FUNCTION_BLOCK FB_L7NHA EXTENDS ZigaLibs_Core.FB_HasInstanceNameAndPath

VAR_INPUT
	bEnable					: BOOL;	// Enable axis
	bReset					: BOOL;	// Reset if an eror is present
	bHalt					: BOOL; // Halts current operation - after setting this to FALSE previous operation is continuoued
	bQuickStop				: BOOL;	// Drive will execute a quick stop
	
	nAcceleration			: UDINT;	// Axis acceleration in UU/s^2
	nDeceleration			: UDINT;	// Axis deceleration in UU/s^
	
	eModeOfOperation		: E_L7NHA_ModeOfOperation;	// Mode of operation
	
	stVelocityCommands		: ST_L7NHA_VelocityCommands;		// Velocity commands when in profile velocity mode
	stPositioningCommands	: ST_L7NHA_PositioningCommands;		// Positioning commands when in profile position mode
	stHomingCommands		: ST_L7NHA_HomingCommands;			// Homing commands when in homing sequence
	stProfileTorqueCommands	: ST_L7NHA_ProfileTorqueCommands;	// Profile torque commands when using Profile Torque mode
	
	fRatedTorque			: REAL; // Rated torque in mNm - required for torque calculation

	stUserUnitParameters	: ST_L7NHA_UserUnitParams;
END_VAR

VAR_OUTPUT
	eAxisState			: E_L7NHA_DriveState;	// Axis state, actual state reported back from drive
	
	eErrorCode			: E_L7NHA_ErrorId;	// Error code, if drive is in fault state
	
	bHomingRequired		: BOOL;	// If homing is required, this flag will be set to true (usually after a power reset)
	
	bMovingPositive		: BOOL;	// Indicating axis is rotating in positive direction
	bMovingNegative		: BOOL;	// Indicating axis is rotating in negative direction
	
	stPositioningStatus	: ST_L7NHA_PositioningStatus;	// Status of the positioning procedure - only valid when in positioning mode
	stHomingStatus		: ST_L7NHA_HomingStatus;		// Status of the homing procedure - only valid when in homing mode
	
	fCalculatedActualTorque	: REAL;
	fCalculatedTargetTorque	: REAL;
	
	eActualModeOfOperation	: E_L7NHA_ModeOfOperation;
	stMotionFeedback		: ST_L7NHA_MotionFeedback;	// Motion feedback from the drive

	stDigitalInputs	:		 ST_L7NHA_DigitalInputs;
	
	bModeOfOperationNotImplemented	: BOOL;	// Will be TRUE if the selected mode of operation is not implemented (axis has to be in enabled state for this flag to be valid!)
END_VAR

// Local variables
VAR
	eAxisStateInternal		: E_L7NHA_DriveState;
	stDataToDriveInternal	: ST_L7NHA_DataToDrive;
	TonCommandTimeout		: Tc2_Standard.TON := (PT := T#1S);
	RtrigMoveToPosition		: Tc2_Standard.R_TRIG;
	RtrigStartHoming		: Tc2_Standard.R_TRIG;
	nPreviousPosition		: DINT;
	RtrigResetTrigger		: Tc2_Standard.R_TRIG;
	RtrigHomingFinished		: Tc2_Standard.R_TRIG;
	TonMotorMovingStatusValid	: Tc2_Standard.TON;
	RtrigModeOfOperationNotImplemented	: Tc2_Standard.R_TRIG;
	eModeOfOpereationOld		: E_L7NHA_ModeOfOperation;
	_logger					: REFERENCE TO ZigaLibs_Logging.I_Logger;
	_sb						: ZigaLibs_Core.FB_StringBuilder;
END_VAR

// IO
VAR
	stDataFromDrive	AT %I* : ST_L7NHA_DataFromDrive;
	stDataToDrive	AT %Q* : ST_L7NHA_DataToDrive;
	stEthercatInfo	AT %I* : ST_L7NHA_EthercatData;
END_VAR

// Sometimes axis wont go to enabled - in that case a timeout should be triggered
TonCommandTimeout(in := eAxisStateInternal = E_L7NHA_DriveState.OPERATION_ENABLED);
// Reset triggering
RtrigResetTrigger(CLK := bReset);


// Abs encoder value is not valid if bit 14 is FALSE (homing has not been completed yet after a power reset/encoder error)
bHomingRequired := stDataFromDrive.StatusWord.14 = FALSE;

// Calling halt will overwrite this - to enable automatic clearing, setting it to false by default
stDataToDriveInternal.ControlWord.8 := FALSE;

// State machine based on the drive's feedback
eAxisStateInternal := THIS^.GetDriveState();

bModeOfOperationNotImplemented := FALSE;
		
// State machine based on actual state reported back from the drive
CASE eAxisStateInternal OF
	E_L7NHA_DriveState.SWITCH_ON_DISABLED:	
		IF bEnable THEN
			Shutdown();
		ELSE
			DisableVoltage();
		END_IF
	
	E_L7NHA_DriveState.READY_TO_SWITCH_ON:
		IF NOT TonCommandTimeout.Q THEN
			SwitchOnEnableOperation();
		END_IF
		
	E_L7NHA_DriveState.OPERATION_ENABLED:
		TonCommandTimeout.IN := FALSE;
		SwitchOnEnableOperation();

		// Execute different mode based on mode of operation setting
		CASE eModeOfOperation OF
			E_L7NHA_ModeOfOperation.PROFILE_POSITION:
				ProfilePosition();
				
			E_L7NHA_ModeOfOperation.PROFILE_VELOCITY:
				ProfileVelocity();
				
			E_L7NHA_ModeOfOperation.HOMING:
				Homing();
				
			E_L7NHA_ModeOfOperation.PROFILE_TORQUE:
				ProfileTorque();
				
			ELSE
				bModeOfOperationNotImplemented := TRUE;
				IF eModeOfOperation <> eModeOfOpereationOld THEN
					IF __ISVALIDREF(_logger) THEN
						_logger.LogError(_sb.Reset()
							.AddString('L7NHA axis ')
							.AddWithDblQuotationMarks(THIS^.InstanceName)
							.AddString(': Mode of operation is not supported! Selected mode is ')
							.AddWithDblQuotationMarks(TO_STRING(eModeOfOperation)));
					END_IF
				END_IF
		END_CASE
		
	E_L7NHA_DriveState.FAULT:
		IF RtrigResetTrigger.Q THEN
			FaultReset();
		ELSE
			stDataToDriveInternal.ControlWord.7 := FALSE;
		END_IF
	
END_CASE

// Override any command if enable is false (transitioning states) - exception is fault, where reset needs to be sent
IF NOT bEnable AND eAxisStateInternal <> E_L7NHA_DriveState.FAULT THEN
	DisableVoltage();
END_IF

// Halt - has a different meaning in PP,PV or homing 
// Usally it "pauses" the current procedure and after halt is set to FALSE drive will proceed where it left off
IF bHalt THEN
	Halt();
END_IF

// Quick stop
IF bQuickStop THEN
	stDataToDriveInternal.ControlWord.1 := bQuickStop;
	stDataToDriveInternal.ControlWord.2 := NOT bQuickStop;
END_IF

// Setting acceleration/deceleration always
stDataToDriveInternal.ProfileAcceleration := nAcceleration;
stDataToDriveInternal.ProfileDeceleration := nDeceleration;

// Mode of operation
stDataToDriveInternal.ModeOfOperation := eModeOfOperation;


// =======================================================================
// ==================== SETTING FB OUTPUTS ===============================
// =======================================================================

// Axis state
eAxisState := eAxisStateInternal;

// Overwriting status for positioning/homing if not in that mode
// Clear homing status if not in that mode
IF eModeOfOperation <> E_L7NHA_ModeOfOperation.HOMING THEN
	MEMSET(
		destAddr := ADR(stHomingStatus),
		n := SIZEOF(stHomingStatus),
		fillByte := 0);
END_IF
 
// Clear positioning status if not in that mode
IF eModeOfOperation <> E_L7NHA_ModeOfOperation.PROFILE_POSITION THEN
	MEMSET(
		destAddr := ADR(stPositioningStatus),
		n := SIZEOF(stPositioningStatus),
		fillByte := 0);
END_IF

// Motion status
TonMotorMovingStatusValid(
	IN := nPreviousPosition <> stDataFromDrive.MotionFeedback.ActualPosition,
	PT := T#30MS);

bMovingPositive := (nPreviousPosition < stDataFromDrive.MotionFeedback.ActualPosition) AND TonMotorMovingStatusValid.Q;
bMovingNegative := (nPreviousPosition > stDataFromDrive.MotionFeedback.ActualPosition) AND TonMotorMovingStatusValid.Q;
nPreviousPosition := stDataFromDrive.MotionFeedback.ActualPosition;

// Digital inputs mapping
stDigitalInputs.NOT_SW := stDataFromDrive.DigitalInputs.0;
stDigitalInputs.POT_SW := stDataFromDrive.DigitalInputs.1;
stDigitalInputs.DI1_OPEN := stDataFromDrive.DigitalInputs.16;
stDigitalInputs.DI2_OPEN := stDataFromDrive.DigitalInputs.17;
stDigitalInputs.DI3_OPEN := stDataFromDrive.DigitalInputs.18;
stDigitalInputs.DI4_OPEN := stDataFromDrive.DigitalInputs.19;
stDigitalInputs.DI5_OPEN := stDataFromDrive.DigitalInputs.20;
stDigitalInputs.DI6_OPEN := stDataFromDrive.DigitalInputs.21;
stDigitalInputs.DI7_OPEN := stDataFromDrive.DigitalInputs.22;
stDigitalInputs.DI8_OPEN := stDataFromDrive.DigitalInputs.23;
stDigitalInputs.STO_OPEN := stDataFromDrive.DigitalInputs.31;

// Error code
IF eErrorCode <> stDataFromDrive.ErrorCode THEN
	IF __ISVALIDREF(_logger) THEN
		IF stDataFromDrive.ErrorCode = E_L7NHA_ErrorId.NO_ERROR THEN
			_logger.LogInfo(_sb.Reset()
				.AddString('L7NHA axis ')
				.AddWithDblQuotationMarks(THIS^.InstanceName)
				.AddString(' error no longer active.')
				.Create());
		ELSE
			_logger.LogError(_sb.Reset()
				.AddString('L7NHA axis ')
				.AddWithDblQuotationMarks(THIS^.InstanceName)
				.AddString(' error active! Error code: ')
				.AddString(TO_STRING(stDataFromDrive.ErrorCode))
				.AddString(' !')
				.Create());
		END_IF
	END_IF
END_IF

eErrorCode := stDataFromDrive.ErrorCode;

// Motion feedback from drive
stMotionFeedback := stDataFromDrive.MotionFeedback;
// Convert position/velocity to custom units

stMotionFeedback := stDataFromDrive.MotionFeedback;

fCalculatedActualTorque := CalculateTorque(fRatedTorque := fRatedTorque, nDriveTorqueFeedback := stDataFromDrive.MotionFeedback.ActualTorque);
fCalculatedTargetTorque := CalculateTorque(fRatedTorque := fRatedTorque, nDriveTorqueFeedback := stDataFromDrive.MotionFeedback.TargetTorque);

// Actual mode of operation, read from the drive
eActualModeOfOperation := stDataFromDrive.ModeOfOperation;

eModeOfOpereationOld := eModeOfOperation;

// =======================================================================
// ==================== SETTING OUTPUT STRUCTURE TO DRIVE ================
// =======================================================================
stDataToDrive := stDataToDriveInternal;

METHOD PRIVATE CalculateTorque : REAL
VAR_INPUT
	fRatedTorque 			: REAL; // Rated torque in mNm
	nDriveTorqueFeedback 	: INT;	// Drives feedback (0.1% increments, -100%...+100%)
END_VAR
CalculateTorque := fRatedTorque * TO_REAL(nDriveTorqueFeedback);
END_METHOD

METHOD PRIVATE DisableVoltage
stDataToDriveInternal.controlWord := 0;
END_METHOD

METHOD PRIVATE EnableOperation
stDataToDriveInternal.controlWord.0 := 0;
stDataToDriveInternal.controlWord.1 := 1;
stDataToDriveInternal.controlWord.2 := 1;
stDataToDriveInternal.controlWord.3 := 0;
stDataToDriveInternal.controlWord.4 := 0;
stDataToDriveInternal.controlWord.5 := 0;
stDataToDriveInternal.controlWord.6 := 0;
stDataToDriveInternal.controlWord.7 := 0;
END_METHOD

METHOD PRIVATE FaultReset
IF stDataToDriveInternal.controlWord.7 = 0 THEN
	stDataToDriveInternal.controlWord.7 := 1;
	stDataToDriveInternal.controlWord.0 := 0;
	stDataToDriveInternal.controlWord.1 := 0;
	stDataToDriveInternal.controlWord.2 := 0;
	stDataToDriveInternal.controlWord.3 := 0;
END_IF
END_METHOD

METHOD FB_init : BOOL
VAR_INPUT
	bInitRetains : BOOL; // if TRUE, the retain variables are initialized (warm start / cold start)
	bInCopyCode : BOOL;  // if TRUE, the instance afterwards gets moved into the copy code (online change)
	logger		: REFERENCE TO ZigaLibs_Logging.I_Logger; // If you do not want logging, simply set this variable to 0, internal checks will ommit any logging.		
END_VAR
_logger REF= logger;
END_METHOD

// Converts status word to a readable drive state enum
METHOD PRIVATE GetDriveState : E_L7NHA_DriveState
//================ SWITCH_ON_DISABLED =====================
IF stDataFromDrive.StatusWord.0 = FALSE AND
    stDataFromDrive.StatusWord.1 = FALSE AND
    stDataFromDrive.StatusWord.2 = FALSE AND
    stDataFromDrive.StatusWord.3 = FALSE AND
    stDataFromDrive.StatusWord.5 = TRUE AND 
    stDataFromDrive.StatusWord.6 = TRUE
THEN
	GetDriveState := E_L7NHA_DriveState.SWITCH_ON_DISABLED;

//================ READY_TO_SWITCH_ON =====================	
ELSIF stDataFromDrive.StatusWord.0 = TRUE AND
   	   stDataFromDrive.StatusWord.1 = FALSE AND
       stDataFromDrive.StatusWord.2 = FALSE AND
       stDataFromDrive.StatusWord.3 = FALSE AND
       stDataFromDrive.StatusWord.5 = TRUE AND 
       stDataFromDrive.StatusWord.6 = FALSE
THEN
	GetDriveState := E_L7NHA_DriveState.READY_TO_SWITCH_ON;	

//================ SWITCHED_ON ==========================	
ELSIF stDataFromDrive.StatusWord.0 = TRUE AND
   	   stDataFromDrive.StatusWord.1 = TRUE AND
       stDataFromDrive.StatusWord.2 = FALSE AND
       stDataFromDrive.StatusWord.3 = FALSE AND
       stDataFromDrive.StatusWord.5 = TRUE AND 
       stDataFromDrive.StatusWord.6 = FALSE
THEN
	GetDriveState := E_L7NHA_DriveState.SWITCHED_ON;

//================ OPERATION_ENABLED =====================	
ELSIF stDataFromDrive.StatusWord.0 = TRUE AND
   	   stDataFromDrive.StatusWord.1 = TRUE AND
       stDataFromDrive.StatusWord.2 = TRUE AND
       stDataFromDrive.StatusWord.3 = FALSE AND
       stDataFromDrive.StatusWord.5 = TRUE AND 
       stDataFromDrive.StatusWord.6 = FALSE
THEN
	GetDriveState := E_L7NHA_DriveState.OPERATION_ENABLED;

//================ FAULT_REACTION_ACTIVE =====================		
ELSIF stDataFromDrive.StatusWord.0 = TRUE AND
   	   stDataFromDrive.StatusWord.1 = TRUE AND
       stDataFromDrive.StatusWord.2 = TRUE AND
       stDataFromDrive.StatusWord.3 = TRUE AND
       stDataFromDrive.StatusWord.5 = TRUE AND 
       stDataFromDrive.StatusWord.6 = FALSE
THEN
	GetDriveState := E_L7NHA_DriveState.FAULT_REACTION_ACTIVE;

//================ FAULT =====================	
ELSIF  stDataFromDrive.StatusWord.0 = FALSE AND
   	   stDataFromDrive.StatusWord.1 = FALSE AND
       stDataFromDrive.StatusWord.2 = FALSE AND
       stDataFromDrive.StatusWord.3 = TRUE AND 
       stDataFromDrive.StatusWord.6 = FALSE
THEN
	GetDriveState := E_L7NHA_DriveState.FAULT;				
END_IF
END_METHOD

// Halts the axis for as long as called
METHOD PRIVATE Halt : BOOL
VAR_INPUT
END_VAR
stDataToDriveInternal.ControlWord.8 := TRUE;
END_METHOD

ACTION Homing:
// Set the status of homing

// Hooming is in progress
stHomingStatus.InProgress := 
stDataFromDrive.StatusWord.10 = FALSE AND
stDataFromDrive.StatusWord.12 = FALSE AND
stDataFromDrive.StatusWord.13 = FALSE;

// Homing is not started
stHomingStatus.NotStarted := 
stDataFromDrive.StatusWord.10 = TRUE AND
stDataFromDrive.StatusWord.12 = FALSE AND
stDataFromDrive.StatusWord.13 = FALSE;	

// Target not reached	
stHomingStatus.TargetNotReached := 
stDataFromDrive.StatusWord.10 = FALSE AND
stDataFromDrive.StatusWord.12 = TRUE AND
stDataFromDrive.StatusWord.13 = FALSE;

// Homing completed
stHomingStatus.Completed := 
stDataFromDrive.StatusWord.10 = TRUE AND
stDataFromDrive.StatusWord.12 = TRUE AND
stDataFromDrive.StatusWord.13 = FALSE;

// Error - speed is not zero ????
stHomingStatus.ErrorSpeedNotZero := 
stDataFromDrive.StatusWord.10 = FALSE AND
stDataFromDrive.StatusWord.12 = FALSE AND
stDataFromDrive.StatusWord.13 = TRUE;

// Error - speed is zero ????
stHomingStatus.ErrorSpeedIsZero := 
stDataFromDrive.StatusWord.10 = TRUE AND
stDataFromDrive.StatusWord.12 = FALSE AND
stDataFromDrive.StatusWord.13 = TRUE;


RtrigStartHoming(CLK := stHomingCommands.Start);	
IF stHomingCommands.Enable = FALSE THEN
	stDataToDriveInternal.ControlWord.4 := FALSE;
ELSIF RtrigStartHoming.Q THEN
	stDataToDriveInternal.ControlWord.4 := TRUE;
END_IF

RtrigHomingFinished(CLK := stHomingStatus.Completed);
IF RtrigHomingFinished.Q THEN
	stDataToDriveInternal.ControlWord.4 := FALSE;
END_IF
END_ACTION

ACTION ProfilePosition:
// Positioning is only allowed if homing has been executed
IF NOT bHomingRequired THEN					
	// Set maximum velocity
	stDataToDriveInternal.MaximumProfileVelocity := stPositioningCommands.MaxVelocity;
	
	// Update target immediately - bit 5 is TRUE
	stDataToDriveInternal.ControlWord.5 := TRUE;
	
	// Trigger immediate update of setpoint by toggling the bit
	IF stPositioningCommands.EnablePositioning THEN
		// Toggling of bit 4 will execute the changes as soon as they are written
		IF stPositioningCommands.ImmediatePositioning THEN
			stDataToDriveInternal.ControlWord.4 := NOT stDataToDriveInternal.ControlWord.4;
			stDataToDriveInternal.ProfileVelocity := stPositioningCommands.VelocitySetpoint;
			stDataToDriveInternal.TargetPosition := stPositioningCommands.TargetPosition;
		ELSE
			// Bit 4 is only set for 1 cycle when requested by the GoToPosition trigger
			stDataToDriveInternal.ControlWord.4 := FALSE;
			// Sending values only on triger of GoToPosition property
			RtrigMoveToPosition(CLK := stPositioningCommands.GoToPosition);
			IF RtrigMoveToPosition.Q THEN
				stDataToDriveInternal.ControlWord.4 := TRUE;
				stDataToDriveInternal.ProfileVelocity := stPositioningCommands.VelocitySetpoint;
				stDataToDriveInternal.TargetPosition := stPositioningCommands.TargetPosition;
			END_IF
		END_IF
	ELSE
		Halt();
	END_IF
	
	// Positioning status from drive
	stPositioningStatus.TargetPositionReached := stDataFromDrive.StatusWord.10;
	stPositioningStatus.SetpointAcknowledged := stDataFromDrive.StatusWord.12;
	stPositioningStatus.PositionalError := stDataFromDrive.StatusWord.13;
ELSE
	// If homing has not been executed, halt axis
	Halt();
END_IF
END_ACTION

ACTION ProfileTorque:
stDataToDriveInternal.TorqueCommands := stProfileTorqueCommands;
END_ACTION

ACTION ProfileVelocity:
// Velocity mode is very simple - just send out the speed setpoint
stDataToDriveInternal.TargetVelocity := stVelocityCommands.VelocitySetpoint;
END_ACTION

METHOD PRIVATE Shutdown
stDataToDriveInternal.controlWord.0 := 0;
stDataToDriveInternal.controlWord.1 := 1;
stDataToDriveInternal.controlWord.2 := 1;
stDataToDriveInternal.controlWord.7 := 0;
END_METHOD

METHOD PRIVATE SwitchOn
stDataToDriveInternal.controlWord.0 := 1;
stDataToDriveInternal.controlWord.1 := 1;
stDataToDriveInternal.controlWord.2 := 1;
stDataToDriveInternal.controlWord.3 := 0;
END_METHOD

METHOD PRIVATE SwitchOnEnableOperation
stDataToDriveInternal.controlWord.0 := 1;
stDataToDriveInternal.controlWord.1 := 1;
stDataToDriveInternal.controlWord.2 := 1;
stDataToDriveInternal.controlWord.3 := 1;
END_METHOD

END_FUNCTION_BLOCK

(* stored: Version 1.1.0.1
   POU FB_L7NHA: Id {eb8da92c-d07d-4e07-b97c-65d4e28a779c}, SpecialFunc None
   Folder Commands: Id {467138cf-83df-4b25-81eb-d9f74aa509c2}
   Folder Modes of operation: Id {d85e02d1-cf3b-4d2d-8776-69be560bc17b}
   Method CalculateTorque: Id {d7606ade-1dc1-4560-9428-c0c8f7068a54}
   Method DisableVoltage: Id {eceaee80-559a-4970-8177-40812eb33d5c}
   Method EnableOperation: Id {90edd31e-d8ca-43a5-bf52-1210d9b5fe6d}
   Method FaultReset: Id {6305dea6-2e84-49e8-8aa5-8326e4ba6a8d}
   Method FB_init: Id {b81cf2d5-c33a-0036-37f3-b25fb7853eb3}
   Method GetDriveState: Id {00293757-5568-4439-9381-8a12fdd5238b}
   Method Halt: Id {989bc803-d6d9-4e40-9538-4cf8a6da3fd4}
   Action Homing: Id {204e4768-faa4-4836-ad0f-0a11eb054788}
   Action ProfilePosition: Id {8f7b2db0-3f6c-4ac6-bcc4-ce2161b443d1}
   Action ProfileTorque: Id {0456e217-0bbc-0ad2-0101-17fd02b1c5b6}
   Action ProfileVelocity: Id {ca6e31c0-beef-44b0-8925-04e717abb05a}
   Method Shutdown: Id {251a3e90-0e6d-48ef-bfa4-28d18e2d967a}
   Method SwitchOn: Id {5f069525-2bd5-4c50-86b6-9baad3ae4272}
   Method SwitchOnEnableOperation: Id {f58b2024-f506-4b25-9cd7-3c25ec539a9b} *)
